PROGRAM PRG_Environment
VAR
END_VAR

// DREAM KB Internal RTDs
    GVL_M4K4_RTD.nM4K4_Chin_Left_RTD();
    GVL_M4K4_RTD.nM4K4_Chin_Right_RTD();
    GVL_M4K4_RTD.nM4K4_Chin_Tail_RTD();

    GVL_M5K4_RTD.nM5K4_Chin_Left_RTD();
    GVL_M5K4_RTD.nM5K4_Chin_Right_RTD();
    GVL_M5K4_RTD.nM5K4_Chin_Tail_RTD();

END_PROGRAM

(* stored: Version 1.1.0.1, ProductVersion 3.1.4024.12
   POU PRG_Environment: Id {d7d13681-7518-4597-8191-c148d0adcca3}, SpecialFunc None *)
